(* IEC 61131-3 sources: rk/stdlib, 15 files *)

(* ---- Arrays.st ---- *)
/*
Array functions.

`LOWER_BOUND` and `UPPER_BOUND` read the bounds of an array. They take an
array of any type and any number of dimensions, so a FUNCTION with an
`ARRAY[*]` parameter can walk whatever array its caller passed.

`GET_DWORD_BE` and its siblings read a WORD, a DWORD, an LWORD, a REAL or an
LREAL out of an array of bytes, at a subscript of that array, in big-endian
(`_BE`) or little-endian (`_LE`) order. `PUT_DWORD_BE` and its siblings
write one. A position whose bytes are not all in the array faults, as any
subscript past its bounds does.
*/
NAMESPACE Std.Arrays

	/* Returns the lower bound of dimension `DIM` of `ARR`.

	   Dimensions are numbered from 1. A `DIM` outside them raises.

	   # Examples

	   ```iecst
	   FOR i := LOWER_BOUND(values, 1) TO UPPER_BOUND(values, 1) DO
	       total := total + values[i];
	   END_FOR;
	   ```
	*/
	FUNCTION LOWER_BOUND: DINT
		VAR_INPUT
			ARR: ARRAY[*];
			DIM: DINT;
		END_VAR
		VAR
			dimensions: DINT;
		END_VAR

		{wasm 'array.dimensions' (params ARR) (result dimensions)}
		IF DIM < 1 OR DIM > dimensions THEN
			__RAISE('array dimension out of range');
		END_IF
		{wasm 'array.lower_bound' (params ARR DIM) (result LOWER_BOUND)}
	END_FUNCTION

	/* Returns the upper bound of dimension `DIM` of `ARR`.

	   Dimensions are numbered from 1. A `DIM` outside them raises.

	   # Examples

	   ```iecst
	   // m : ARRAY[1..3, 0..9] OF REAL
	   rows := UPPER_BOUND(m, 1) - LOWER_BOUND(m, 1) + 1;     // 3
	   columns := UPPER_BOUND(m, 2) - LOWER_BOUND(m, 2) + 1;  // 10
	   ```
	*/
	FUNCTION UPPER_BOUND: DINT
		VAR_INPUT
			ARR: ARRAY[*];
			DIM: DINT;
		END_VAR
		VAR
			dimensions: DINT;
		END_VAR

		{wasm 'array.dimensions' (params ARR) (result dimensions)}
		IF DIM < 1 OR DIM > dimensions THEN
			__RAISE('array dimension out of range');
		END_IF
		{wasm 'array.upper_bound' (params ARR DIM) (result UPPER_BOUND)}
	END_FUNCTION

	/* Returns the value whose bytes are in `buf` from `pos` on, in big-endian
	   order: the most significant at `pos`.

	   # Examples

	   ```iecst
	   // frame holds 16#12, 16#34, 16#56, 16#78 from its subscript 0 on
	   d := GET_DWORD_BE(frame, 0);  // DWORD#16#12345678
	   w := GET_WORD_BE(frame, 2);   // WORD#16#5678
	   ```
	*/
	FUNCTION GET_WORD_BE: WORD
		VAR_IN_OUT
			buf: ARRAY[*] OF BYTE;
		END_VAR
		VAR_INPUT
			pos: DINT;
		END_VAR
		GET_WORD_BE.%B1 := buf[pos];
		GET_WORD_BE.%B0 := buf[pos + 1];
	END_FUNCTION

	FUNCTION GET_DWORD_BE: DWORD
		VAR_IN_OUT
			buf: ARRAY[*] OF BYTE;
		END_VAR
		VAR_INPUT
			pos: DINT;
		END_VAR
		GET_DWORD_BE.%B3 := buf[pos];
		GET_DWORD_BE.%B2 := buf[pos + 1];
		GET_DWORD_BE.%B1 := buf[pos + 2];
		GET_DWORD_BE.%B0 := buf[pos + 3];
	END_FUNCTION

	FUNCTION GET_LWORD_BE: LWORD
		VAR_IN_OUT
			buf: ARRAY[*] OF BYTE;
		END_VAR
		VAR_INPUT
			pos: DINT;
		END_VAR
		GET_LWORD_BE.%B7 := buf[pos];
		GET_LWORD_BE.%B6 := buf[pos + 1];
		GET_LWORD_BE.%B5 := buf[pos + 2];
		GET_LWORD_BE.%B4 := buf[pos + 3];
		GET_LWORD_BE.%B3 := buf[pos + 4];
		GET_LWORD_BE.%B2 := buf[pos + 5];
		GET_LWORD_BE.%B1 := buf[pos + 6];
		GET_LWORD_BE.%B0 := buf[pos + 7];
	END_FUNCTION

	FUNCTION GET_REAL_BE: REAL
		VAR_IN_OUT
			buf: ARRAY[*] OF BYTE;
		END_VAR
		VAR_INPUT
			pos: DINT;
		END_VAR
		VAR
			v: DWORD;
		END_VAR
		v := GET_DWORD_BE(buf, pos);
		{wasm 'f32.reinterpret_i32' (params v) (result GET_REAL_BE)}
	END_FUNCTION

	FUNCTION GET_LREAL_BE: LREAL
		VAR_IN_OUT
			buf: ARRAY[*] OF BYTE;
		END_VAR
		VAR_INPUT
			pos: DINT;
		END_VAR
		VAR
			v: LWORD;
		END_VAR
		v := GET_LWORD_BE(buf, pos);
		{wasm 'f64.reinterpret_i64' (params v) (result GET_LREAL_BE)}
	END_FUNCTION

	/* Returns the value whose bytes are in `buf` from `pos` on, in
	   little-endian order: the least significant at `pos`.

	   # Examples

	   ```iecst
	   // frame holds 16#12, 16#34, 16#56, 16#78 from its subscript 0 on
	   d := GET_DWORD_LE(frame, 0);  // DWORD#16#78563412
	   ```
	*/
	FUNCTION GET_WORD_LE: WORD
		VAR_IN_OUT
			buf: ARRAY[*] OF BYTE;
		END_VAR
		VAR_INPUT
			pos: DINT;
		END_VAR
		GET_WORD_LE.%B0 := buf[pos];
		GET_WORD_LE.%B1 := buf[pos + 1];
	END_FUNCTION

	FUNCTION GET_DWORD_LE: DWORD
		VAR_IN_OUT
			buf: ARRAY[*] OF BYTE;
		END_VAR
		VAR_INPUT
			pos: DINT;
		END_VAR
		GET_DWORD_LE.%B0 := buf[pos];
		GET_DWORD_LE.%B1 := buf[pos + 1];
		GET_DWORD_LE.%B2 := buf[pos + 2];
		GET_DWORD_LE.%B3 := buf[pos + 3];
	END_FUNCTION

	FUNCTION GET_LWORD_LE: LWORD
		VAR_IN_OUT
			buf: ARRAY[*] OF BYTE;
		END_VAR
		VAR_INPUT
			pos: DINT;
		END_VAR
		GET_LWORD_LE.%B0 := buf[pos];
		GET_LWORD_LE.%B1 := buf[pos + 1];
		GET_LWORD_LE.%B2 := buf[pos + 2];
		GET_LWORD_LE.%B3 := buf[pos + 3];
		GET_LWORD_LE.%B4 := buf[pos + 4];
		GET_LWORD_LE.%B5 := buf[pos + 5];
		GET_LWORD_LE.%B6 := buf[pos + 6];
		GET_LWORD_LE.%B7 := buf[pos + 7];
	END_FUNCTION

	FUNCTION GET_REAL_LE: REAL
		VAR_IN_OUT
			buf: ARRAY[*] OF BYTE;
		END_VAR
		VAR_INPUT
			pos: DINT;
		END_VAR
		VAR
			v: DWORD;
		END_VAR
		v := GET_DWORD_LE(buf, pos);
		{wasm 'f32.reinterpret_i32' (params v) (result GET_REAL_LE)}
	END_FUNCTION

	FUNCTION GET_LREAL_LE: LREAL
		VAR_IN_OUT
			buf: ARRAY[*] OF BYTE;
		END_VAR
		VAR_INPUT
			pos: DINT;
		END_VAR
		VAR
			v: LWORD;
		END_VAR
		v := GET_LWORD_LE(buf, pos);
		{wasm 'f64.reinterpret_i64' (params v) (result GET_LREAL_LE)}
	END_FUNCTION

	/* Writes the bytes of `value` into `buf` from `pos` on, in big-endian
	   order: the most significant at `pos`.

	   # Examples

	   ```iecst
	   PUT_DWORD_BE(frame, 0, DWORD#16#12345678);  // 16#12, 16#34, 16#56, 16#78
	   PUT_REAL_BE(frame, 4, REAL#1.0);            // 16#3F, 16#80, 16#00, 16#00
	   ```
	*/
	FUNCTION PUT_WORD_BE
		VAR_IN_OUT
			buf: ARRAY[*] OF BYTE;
		END_VAR
		VAR_INPUT
			pos: DINT;
			value: WORD;
		END_VAR
		buf[pos] := value.%B1;
		buf[pos + 1] := value.%B0;
	END_FUNCTION

	FUNCTION PUT_DWORD_BE
		VAR_IN_OUT
			buf: ARRAY[*] OF BYTE;
		END_VAR
		VAR_INPUT
			pos: DINT;
			value: DWORD;
		END_VAR
		buf[pos] := value.%B3;
		buf[pos + 1] := value.%B2;
		buf[pos + 2] := value.%B1;
		buf[pos + 3] := value.%B0;
	END_FUNCTION

	FUNCTION PUT_LWORD_BE
		VAR_IN_OUT
			buf: ARRAY[*] OF BYTE;
		END_VAR
		VAR_INPUT
			pos: DINT;
			value: LWORD;
		END_VAR
		buf[pos] := value.%B7;
		buf[pos + 1] := value.%B6;
		buf[pos + 2] := value.%B5;
		buf[pos + 3] := value.%B4;
		buf[pos + 4] := value.%B3;
		buf[pos + 5] := value.%B2;
		buf[pos + 6] := value.%B1;
		buf[pos + 7] := value.%B0;
	END_FUNCTION

	FUNCTION PUT_REAL_BE
		VAR_IN_OUT
			buf: ARRAY[*] OF BYTE;
		END_VAR
		VAR_INPUT
			pos: DINT;
			value: REAL;
		END_VAR
		VAR
			v: DWORD;
		END_VAR
		{wasm 'i32.reinterpret_f32' (params value) (result v)}
		PUT_DWORD_BE(buf, pos, v);
	END_FUNCTION

	FUNCTION PUT_LREAL_BE
		VAR_IN_OUT
			buf: ARRAY[*] OF BYTE;
		END_VAR
		VAR_INPUT
			pos: DINT;
			value: LREAL;
		END_VAR
		VAR
			v: LWORD;
		END_VAR
		{wasm 'i64.reinterpret_f64' (params value) (result v)}
		PUT_LWORD_BE(buf, pos, v);
	END_FUNCTION

	/* Writes the bytes of `value` into `buf` from `pos` on, in little-endian
	   order: the least significant at `pos`.

	   # Examples

	   ```iecst
	   PUT_DWORD_LE(frame, 0, DWORD#16#12345678);  // 16#78, 16#56, 16#34, 16#12
	   ```
	*/
	FUNCTION PUT_WORD_LE
		VAR_IN_OUT
			buf: ARRAY[*] OF BYTE;
		END_VAR
		VAR_INPUT
			pos: DINT;
			value: WORD;
		END_VAR
		buf[pos] := value.%B0;
		buf[pos + 1] := value.%B1;
	END_FUNCTION

	FUNCTION PUT_DWORD_LE
		VAR_IN_OUT
			buf: ARRAY[*] OF BYTE;
		END_VAR
		VAR_INPUT
			pos: DINT;
			value: DWORD;
		END_VAR
		buf[pos] := value.%B0;
		buf[pos + 1] := value.%B1;
		buf[pos + 2] := value.%B2;
		buf[pos + 3] := value.%B3;
	END_FUNCTION

	FUNCTION PUT_LWORD_LE
		VAR_IN_OUT
			buf: ARRAY[*] OF BYTE;
		END_VAR
		VAR_INPUT
			pos: DINT;
			value: LWORD;
		END_VAR
		buf[pos] := value.%B0;
		buf[pos + 1] := value.%B1;
		buf[pos + 2] := value.%B2;
		buf[pos + 3] := value.%B3;
		buf[pos + 4] := value.%B4;
		buf[pos + 5] := value.%B5;
		buf[pos + 6] := value.%B6;
		buf[pos + 7] := value.%B7;
	END_FUNCTION

	FUNCTION PUT_REAL_LE
		VAR_IN_OUT
			buf: ARRAY[*] OF BYTE;
		END_VAR
		VAR_INPUT
			pos: DINT;
			value: REAL;
		END_VAR
		VAR
			v: DWORD;
		END_VAR
		{wasm 'i32.reinterpret_f32' (params value) (result v)}
		PUT_DWORD_LE(buf, pos, v);
	END_FUNCTION

	FUNCTION PUT_LREAL_LE
		VAR_IN_OUT
			buf: ARRAY[*] OF BYTE;
		END_VAR
		VAR_INPUT
			pos: DINT;
			value: LREAL;
		END_VAR
		VAR
			v: LWORD;
		END_VAR
		{wasm 'i64.reinterpret_f64' (params value) (result v)}
		PUT_LWORD_LE(buf, pos, v);
	END_FUNCTION

	NAMESPACE Test
		USING Std.Unit

		{test}
		FUNCTION test_bounds_of_one_dimension
			VAR
				a: ARRAY[1..10] OF INT;
			END_VAR
			ASSERT(LOWER_BOUND(a, 1) = 1 AND UPPER_BOUND(a, 1) = 10);
		END_FUNCTION

		{test}
		FUNCTION test_bounds_of_each_dimension
			VAR
				a: ARRAY[1..20, -2..2] OF INT;
			END_VAR
			ASSERT(LOWER_BOUND(a, 1) = 1 AND UPPER_BOUND(a, 1) = 20);
			ASSERT(LOWER_BOUND(a, 2) = -2 AND UPPER_BOUND(a, 2) = 2);
		END_FUNCTION

		{test}
		FUNCTION test_bounds_by_name
			VAR
				a: ARRAY[5..7] OF STRING[4];
			END_VAR
			ASSERT(LOWER_BOUND(ARR := a, DIM := 1) = 5);
			ASSERT(UPPER_BOUND(DIM := 1, ARR := a) = 7);
		END_FUNCTION

		FUNCTION Sum: DINT
			VAR_IN_OUT
				values: ARRAY[*] OF INT;
			END_VAR
			VAR
				i: DINT;
			END_VAR
			FOR i := LOWER_BOUND(values, 1) TO UPPER_BOUND(values, 1) DO
				Sum := Sum + values[i];
			END_FOR
		END_FUNCTION

		{test}
		FUNCTION test_bounds_of_an_array_any_call_binds
			VAR
				a: ARRAY[1..20, -2..2] OF INT := [20(5(1))];
				b: ARRAY[0..2] OF INT := [1, 2, 3];
			END_VAR
			ASSERT(Sum(a[2]) = 5, 'a row of a');
			ASSERT(Sum(b) = 6, 'b');
		END_FUNCTION

		{test}
		FUNCTION test_get_word_be
			VAR b : ARRAY[0..1] OF BYTE := [16#12, 16#34]; END_VAR
			ASSERT_EQ(GET_WORD_BE(b, 0), WORD#16#1234);
		END_FUNCTION

		{test}
		FUNCTION test_get_word_le
			VAR b : ARRAY[0..1] OF BYTE := [16#12, 16#34]; END_VAR
			ASSERT_EQ(GET_WORD_LE(b, 0), WORD#16#3412);
		END_FUNCTION

		{test}
		FUNCTION test_get_dword_at_a_subscript
			VAR b : ARRAY[1..6] OF BYTE := [16#FF, 16#12, 16#34, 16#56, 16#78, 16#FF]; END_VAR
			ASSERT_EQ(GET_DWORD_BE(b, 2), DWORD#16#12345678);
		END_FUNCTION

		{test}
		FUNCTION test_put_dword_be
			VAR b : ARRAY[0..3] OF BYTE; END_VAR
			PUT_DWORD_BE(b, 0, DWORD#16#12345678);
			ASSERT_EQ(b[0], BYTE#16#12);
			ASSERT_EQ(b[3], BYTE#16#78);
		END_FUNCTION

		{test}
		FUNCTION test_put_dword_le
			VAR b : ARRAY[0..3] OF BYTE; END_VAR
			PUT_DWORD_LE(b, 0, DWORD#16#12345678);
			ASSERT_EQ(b[0], BYTE#16#78);
			ASSERT_EQ(b[3], BYTE#16#12);
		END_FUNCTION

		{test}
		FUNCTION test_lword_round_trip
			VAR b : ARRAY[0..9] OF BYTE; END_VAR
			PUT_LWORD_BE(b, 1, LWORD#16#0102030405060708);
			ASSERT_EQ(b[1], BYTE#16#01);
			ASSERT_EQ(b[8], BYTE#16#08);
			ASSERT_EQ(GET_LWORD_BE(b, 1), LWORD#16#0102030405060708);
			ASSERT_EQ(GET_LWORD_LE(b, 1), LWORD#16#0807060504030201);
		END_FUNCTION

		{test}
		FUNCTION test_put_real_be
			VAR b : ARRAY[0..3] OF BYTE; END_VAR
			PUT_REAL_BE(b, 0, REAL#1.0);
			ASSERT_EQ(b[0], BYTE#16#3F);
			ASSERT_EQ(b[1], BYTE#16#80);
			ASSERT_EQ(GET_REAL_BE(b, 0), REAL#1.0);
		END_FUNCTION

		{test}
		FUNCTION test_real_le_round_trip
			VAR b : ARRAY[0..3] OF BYTE; END_VAR
			PUT_REAL_LE(b, 0, REAL#-2.5);
			ASSERT_EQ(b[3], BYTE#16#C0);
			ASSERT_EQ(GET_REAL_LE(b, 0), REAL#-2.5);
		END_FUNCTION

		{test}
		FUNCTION test_put_lreal_be
			VAR b : ARRAY[0..7] OF BYTE; END_VAR
			PUT_LREAL_BE(b, 0, LREAL#1.5);
			ASSERT_EQ(b[0], BYTE#16#3F);
			ASSERT_EQ(b[1], BYTE#16#F8);
			ASSERT_EQ(GET_LREAL_BE(b, 0), LREAL#1.5);
		END_FUNCTION

		{test}
		FUNCTION test_lreal_le_round_trip
			VAR b : ARRAY[0..7] OF BYTE; END_VAR
			PUT_LREAL_LE(b, 0, LREAL#1.5);
			ASSERT_EQ(b[7], BYTE#16#3F);
			ASSERT_EQ(GET_LREAL_LE(b, 0), LREAL#1.5);
		END_FUNCTION
	END_NAMESPACE

END_NAMESPACE

(* ---- Bits.st ---- *)
/*
Bit shift and rotate functions.

Each takes a `BYTE`, `WORD`, `DWORD` or `LWORD` and a count `N`, and returns
the type it was given. The width is that of the type: a `BYTE` is shifted
and rotated within its 8 bits.
*/
NAMESPACE Std.Bits

	/* Returns `IN` shifted left by `N` bits, filling with zeros.

	   Bits shifted past the top of the type are lost. An `N` of the type's width
	   or more gives 0.

	   # Examples

	   ```iecst
	   b := SHL(BYTE#16#0F, 4);    // BYTE#16#F0
	   b := SHL(BYTE#16#FF, 4);    // BYTE#16#F0
	   w := SHL(WORD#16#0001, 8);  // WORD#16#0100
	   b := SHL(BYTE#16#01, 8);    // BYTE#16#00
	   ```
	*/
	FUNCTION SHL: BYTE
		VAR_INPUT
			IN: BYTE;
			N: INT;
		END_VAR
		{wasm IN 'shl' (params IN N) (result SHL)}
	END_FUNCTION

	FUNCTION SHL: WORD
		VAR_INPUT
			IN: WORD;
			N: INT;
		END_VAR
		{wasm IN 'shl' (params IN N) (result SHL)}
	END_FUNCTION

	FUNCTION SHL: DWORD
		VAR_INPUT
			IN: DWORD;
			N: INT;
		END_VAR
		{wasm IN 'shl' (params IN N) (result SHL)}
	END_FUNCTION

	FUNCTION SHL: LWORD
		VAR_INPUT
			IN: LWORD;
			N: INT;
		END_VAR
		{wasm IN 'shl' (params IN N) (result SHL)}
	END_FUNCTION

	/* Returns `IN` shifted right by `N` bits, filling with zeros.

	   An `N` of the type's width or more gives 0.

	   # Examples

	   ```iecst
	   b := SHR(BYTE#16#F0, 4);         // BYTE#16#0F
	   d := SHR(DWORD#16#80000000, 31);  // DWORD#1
	   ```
	*/
	FUNCTION SHR: BYTE
		VAR_INPUT
			IN: BYTE;
			N: INT;
		END_VAR
		{wasm IN 'shr_u' (params IN N) (result SHR)}
	END_FUNCTION

	FUNCTION SHR: WORD
		VAR_INPUT
			IN: WORD;
			N: INT;
		END_VAR
		{wasm IN 'shr_u' (params IN N) (result SHR)}
	END_FUNCTION

	FUNCTION SHR: DWORD
		VAR_INPUT
			IN: DWORD;
			N: INT;
		END_VAR
		{wasm IN 'shr_u' (params IN N) (result SHR)}
	END_FUNCTION

	FUNCTION SHR: LWORD
		VAR_INPUT
			IN: LWORD;
			N: INT;
		END_VAR
		{wasm IN 'shr_u' (params IN N) (result SHR)}
	END_FUNCTION

	/* Returns `IN` rotated left by `N` bits.

	   Bits that leave at the top come back at the bottom. `N` wraps at the type's
	   width, so rotating a `BYTE` by 8 returns it unchanged.

	   # Examples

	   ```iecst
	   b := ROL(BYTE#16#81, 1);  // BYTE#16#03
	   b := ROL(BYTE#16#81, 8);  // BYTE#16#81
	   ```
	*/
	FUNCTION ROL: BYTE
		VAR_INPUT
			IN: BYTE;
			N: INT;
		END_VAR
		{wasm IN 'rotl' (params IN N) (result ROL)}
	END_FUNCTION

	FUNCTION ROL: WORD
		VAR_INPUT
			IN: WORD;
			N: INT;
		END_VAR
		{wasm IN 'rotl' (params IN N) (result ROL)}
	END_FUNCTION

	FUNCTION ROL: DWORD
		VAR_INPUT
			IN: DWORD;
			N: INT;
		END_VAR
		{wasm IN 'rotl' (params IN N) (result ROL)}
	END_FUNCTION

	FUNCTION ROL: LWORD
		VAR_INPUT
			IN: LWORD;
			N: INT;
		END_VAR
		{wasm IN 'rotl' (params IN N) (result ROL)}
	END_FUNCTION

	/* Returns `IN` rotated right by `N` bits.

	   Bits that leave at the bottom come back at the top. `N` wraps at the type's
	   width.

	   # Examples

	   ```iecst
	   b := ROR(BYTE#16#01, 1);  // BYTE#16#80
	   w := ROR(WORD#16#0001, 1);  // WORD#16#8000
	   ```
	*/
	FUNCTION ROR: BYTE
		VAR_INPUT
			IN: BYTE;
			N: INT;
		END_VAR
		{wasm IN 'rotr' (params IN N) (result ROR)}
	END_FUNCTION

	FUNCTION ROR: WORD
		VAR_INPUT
			IN: WORD;
			N: INT;
		END_VAR
		{wasm IN 'rotr' (params IN N) (result ROR)}
	END_FUNCTION

	FUNCTION ROR: DWORD
		VAR_INPUT
			IN: DWORD;
			N: INT;
		END_VAR
		{wasm IN 'rotr' (params IN N) (result ROR)}
	END_FUNCTION

	FUNCTION ROR: LWORD
		VAR_INPUT
			IN: LWORD;
			N: INT;
		END_VAR
		{wasm IN 'rotr' (params IN N) (result ROR)}
	END_FUNCTION

	NAMESPACE Test
		USING Std.Unit

		{test}
		FUNCTION test_shl_byte ASSERT_EQ(SHL(BYTE#16#0F, 4), BYTE#16#F0);
		END_FUNCTION

		{test}
		FUNCTION test_shr_byte ASSERT_EQ(SHR(BYTE#16#F0, 4), BYTE#16#0F);
		END_FUNCTION

		{test}
		FUNCTION test_shl_word ASSERT_EQ(SHL(WORD#16#0001, 8), WORD#16#0100);
		END_FUNCTION

		{test}
		FUNCTION test_shr_word ASSERT_EQ(SHR(WORD#16#0100, 8), WORD#16#0001);
		END_FUNCTION

		{test}
		FUNCTION test_rol_dword ASSERT_EQ(ROL(DWORD#1, 4), DWORD#16);
		END_FUNCTION

		{test}
		FUNCTION test_ror_dword ASSERT_EQ(ROR(DWORD#16, 4), DWORD#1);
		END_FUNCTION

		// --- edge cases ---

		// Shift/rotate by 0 is the identity, independent of storage width.
		{test}
		FUNCTION test_shl_by_zero ASSERT_EQ(SHL(BYTE#16#0F, 0), BYTE#16#0F);
		END_FUNCTION

		{test}
		FUNCTION test_shr_by_zero ASSERT_EQ(SHR(WORD#16#00F0, 0), WORD#16#00F0);
		END_FUNCTION

		{test}
		FUNCTION test_rol_by_zero ASSERT_EQ(ROL(DWORD#16#12345678, 0), DWORD#16#12345678);
		END_FUNCTION

		{test}
		FUNCTION test_ror_by_zero ASSERT_EQ(ROR(DWORD#16#12345678, 0), DWORD#16#12345678);
		END_FUNCTION

		// DWORD is i32-backed, so rotate wraps correctly at 32 bits:
		// the top bit rotated left re-enters at bit 0.
		{test}
		FUNCTION test_rol_dword_wraps_msb ASSERT_EQ(ROL(DWORD#16#80000000, 1), DWORD#1);
		END_FUNCTION

		{test}
		FUNCTION test_ror_dword_wraps_lsb ASSERT_EQ(ROR(DWORD#1, 1), DWORD#16#80000000);
		END_FUNCTION

		// Logical shift right fills with zeros (no sign extension) on a bit type.
		{test}
		FUNCTION test_shr_dword_top_bit ASSERT_EQ(SHR(DWORD#16#80000000, 31), DWORD#1);
		END_FUNCTION

		// --- sub-width masking: shifted-out bits must not leak past the type width ---

		{test}
		FUNCTION test_shl_byte_masks_leak
			ASSERT_EQ(SHL(BYTE#16#FF, 4), BYTE#16#F0, 'SHL BYTE must mask bits above bit 7');
		END_FUNCTION

		{test}
		FUNCTION test_shl_word_masks_leak
			ASSERT_EQ(SHL(WORD#16#FFFF, 8), WORD#16#FF00, 'SHL WORD must mask bits above bit 15');
		END_FUNCTION

		{test}
		FUNCTION test_shl_byte_by_type_width
			ASSERT_EQ(SHL(BYTE#16#01, 8), BYTE#16#00, 'shift by the full type width empties the value');
		END_FUNCTION

		// --- shift count >= width yields 0 (wasm masks the count mod the lane
		// width, so a raw lowering would return the input unchanged) ---

		{test}
		FUNCTION test_shl_dword_by_32
			ASSERT_EQ(SHL(DWORD#1, 32), DWORD#0, 'SHL DWORD by 32 is 0, not a wasm count-mask no-op');
		END_FUNCTION

		{test}
		FUNCTION test_shr_dword_by_32
			ASSERT_EQ(SHR(DWORD#16#80000000, 32), DWORD#0, 'SHR DWORD by 32 is 0');
		END_FUNCTION

		{test}
		FUNCTION test_shr_word_by_32
			ASSERT_EQ(SHR(WORD#16#0001, 32), WORD#0, 'SHR WORD by 32 hits the wasm lane mask');
		END_FUNCTION

		// --- sub-width rotates wrap at the type MSB/LSB, not bit 31 ---

		{test}
		FUNCTION test_rol_byte_wraps_msb
			// The doc example: the wrapped bit re-enters at bit 0, not bit 8.
			ASSERT_EQ(ROL(BYTE#16#81, 1), BYTE#16#03, 'ROL BYTE MSB wraps to bit 0');
		END_FUNCTION

		{test}
		FUNCTION test_ror_byte_wraps_lsb
			ASSERT_EQ(ROR(BYTE#16#01, 1), BYTE#16#80, 'ROR BYTE LSB wraps to bit 7, not bit 31');
		END_FUNCTION

		{test}
		FUNCTION test_rol_word_wraps_msb
			ASSERT_EQ(ROL(WORD#16#8001, 1), WORD#16#0003, 'ROL WORD bit 15 wraps to bit 0');
		END_FUNCTION

		{test}
		FUNCTION test_ror_word_wraps_lsb
			ASSERT_EQ(ROR(WORD#16#0001, 1), WORD#16#8000, 'ROR WORD LSB wraps to bit 15');
		END_FUNCTION

		// Rotate counts are mod the type width.
		{test}
		FUNCTION test_rol_byte_count_mod_width
			ASSERT_EQ(ROL(BYTE#16#81, 0), BYTE#16#81, 'ROL by 0 is identity');
			ASSERT_EQ(ROL(BYTE#16#81, 8), BYTE#16#81, 'ROL by the type width is identity');
			ASSERT_EQ(ROL(BYTE#16#81, 9), BYTE#16#03, 'ROL by 9 = ROL by 1 (mod 8)');
		END_FUNCTION

		// --- LWORD (i64 lane): value, count extension, and 64-bit wraps ---

		{test}
		FUNCTION test_shl_lword_crosses_32
			ASSERT_EQ(SHL(LWORD#1, 32), LWORD#16#0000_0001_0000_0000, 'SHL LWORD must cross the 32-bit line');
		END_FUNCTION

		{test}
		FUNCTION test_shl_lword_by_64
			ASSERT_EQ(SHL(LWORD#1, 64), LWORD#0, 'SHL LWORD by 64 is 0');
		END_FUNCTION

		{test}
		FUNCTION test_shr_lword_top_bit
			ASSERT_EQ(SHR(LWORD#16#8000_0000_0000_0000, 63), LWORD#1, 'logical shift on the i64 lane');
		END_FUNCTION

		{test}
		FUNCTION test_rol_lword_wraps_msb
			ASSERT_EQ(ROL(LWORD#16#8000_0000_0000_0000, 1), LWORD#1, '64-bit MSB wraps to bit 0');
		END_FUNCTION

		{test}
		FUNCTION test_ror_lword_wraps_lsb
			ASSERT_EQ(ROR(LWORD#1, 1), LWORD#16#8000_0000_0000_0000, '64-bit LSB wraps to bit 63');
		END_FUNCTION

		{test}
		FUNCTION test_shr_byte_after_shl_roundtrip
			// SHR on a sub-width type relies on the masked-value invariant.
			ASSERT_EQ(SHR(SHL(BYTE#16#FF, 4), 4), BYTE#16#0F, 'SHL then SHR keeps only surviving bits');
		END_FUNCTION
	END_NAMESPACE
END_NAMESPACE

(* ---- Bytes.st ---- *)
/*
Byte order and BCD.

rk keeps every value in little-endian order, the order of WebAssembly: its
least significant byte at the lowest address. TO_BIG_ENDIAN and
FROM_BIG_ENDIAN reverse the bytes of a value, and TO_LITTLE_ENDIAN and
FROM_LITTLE_ENDIAN return it as it is.

Each takes an integer, a bit string, a REAL, an LREAL, a TIME or an LTIME,
and returns the type it was given. A value of one byte has no order, and is
returned as it is.

BCD stores a number one decimal digit in each 4 bits: WORD#16#0369 is 369.
Its conversions go between a bit string and the unsigned integer of the same
width, from BYTE and USINT to LWORD and ULINT.
*/
NAMESPACE Std.Bytes

	/* Returns `IN` with its bytes in big-endian order, the most significant
	   first: the order a peer reading big-endian data expects.

	   # Examples

	   ```iecst
	   w := TO_BIG_ENDIAN(WORD#16#1234);       // WORD#16#3412
	   d := TO_BIG_ENDIAN(DWORD#16#12345678);  // DWORD#16#78563412
	   b := TO_BIG_ENDIAN(BYTE#16#AB);         // BYTE#16#AB
	   ```
	*/
	FUNCTION TO_BIG_ENDIAN: BYTE
		VAR_INPUT
			IN: BYTE;
		END_VAR
		TO_BIG_ENDIAN := IN;
	END_FUNCTION

	FUNCTION TO_BIG_ENDIAN: SINT
		VAR_INPUT
			IN: SINT;
		END_VAR
		TO_BIG_ENDIAN := IN;
	END_FUNCTION

	FUNCTION TO_BIG_ENDIAN: USINT
		VAR_INPUT
			IN: USINT;
		END_VAR
		TO_BIG_ENDIAN := IN;
	END_FUNCTION

	FUNCTION TO_BIG_ENDIAN: WORD
		VAR_INPUT
			IN: WORD;
		END_VAR
		{wasm IN 'bswap' (params IN) (result TO_BIG_ENDIAN)}
	END_FUNCTION

	FUNCTION TO_BIG_ENDIAN: INT
		VAR_INPUT
			IN: INT;
		END_VAR
		VAR
			swapped: WORD;
		END_VAR
		{wasm IN 'bswap' (params IN) (result swapped)}
		{wasm 'nop' (params swapped) (result TO_BIG_ENDIAN)}
	END_FUNCTION

	FUNCTION TO_BIG_ENDIAN: UINT
		VAR_INPUT
			IN: UINT;
		END_VAR
		{wasm IN 'bswap' (params IN) (result TO_BIG_ENDIAN)}
	END_FUNCTION

	FUNCTION TO_BIG_ENDIAN: DWORD
		VAR_INPUT
			IN: DWORD;
		END_VAR
		{wasm IN 'bswap' (params IN) (result TO_BIG_ENDIAN)}
	END_FUNCTION

	FUNCTION TO_BIG_ENDIAN: DINT
		VAR_INPUT
			IN: DINT;
		END_VAR
		{wasm IN 'bswap' (params IN) (result TO_BIG_ENDIAN)}
	END_FUNCTION

	FUNCTION TO_BIG_ENDIAN: UDINT
		VAR_INPUT
			IN: UDINT;
		END_VAR
		{wasm IN 'bswap' (params IN) (result TO_BIG_ENDIAN)}
	END_FUNCTION

	FUNCTION TO_BIG_ENDIAN: REAL
		VAR_INPUT
			IN: REAL;
		END_VAR
		VAR
			bits: DWORD;
		END_VAR
		{wasm 'i32.reinterpret_f32' (params IN) (result bits)}
		{wasm bits 'bswap' (params bits) (result bits)}
		{wasm 'f32.reinterpret_i32' (params bits) (result TO_BIG_ENDIAN)}
	END_FUNCTION

	FUNCTION TO_BIG_ENDIAN: TIME
		VAR_INPUT
			IN: TIME;
		END_VAR
		{wasm IN 'bswap' (params IN) (result TO_BIG_ENDIAN)}
	END_FUNCTION

	FUNCTION TO_BIG_ENDIAN: LWORD
		VAR_INPUT
			IN: LWORD;
		END_VAR
		{wasm IN 'bswap' (params IN) (result TO_BIG_ENDIAN)}
	END_FUNCTION

	FUNCTION TO_BIG_ENDIAN: LINT
		VAR_INPUT
			IN: LINT;
		END_VAR
		{wasm IN 'bswap' (params IN) (result TO_BIG_ENDIAN)}
	END_FUNCTION

	FUNCTION TO_BIG_ENDIAN: ULINT
		VAR_INPUT
			IN: ULINT;
		END_VAR
		{wasm IN 'bswap' (params IN) (result TO_BIG_ENDIAN)}
	END_FUNCTION

	FUNCTION TO_BIG_ENDIAN: LREAL
		VAR_INPUT
			IN: LREAL;
		END_VAR
		VAR
			bits: LWORD;
		END_VAR
		{wasm 'i64.reinterpret_f64' (params IN) (result bits)}
		{wasm bits 'bswap' (params bits) (result bits)}
		{wasm 'f64.reinterpret_i64' (params bits) (result TO_BIG_ENDIAN)}
	END_FUNCTION

	FUNCTION TO_BIG_ENDIAN: LTIME
		VAR_INPUT
			IN: LTIME;
		END_VAR
		{wasm IN 'bswap' (params IN) (result TO_BIG_ENDIAN)}
	END_FUNCTION

	/* Returns `IN`, whose bytes are in big-endian order, in the order rk
	   computes with.

	   # Examples

	   ```iecst
	   w := FROM_BIG_ENDIAN(WORD#16#3412);     // WORD#16#1234
	   ```
	*/
	FUNCTION FROM_BIG_ENDIAN: BYTE
		VAR_INPUT
			IN: BYTE;
		END_VAR
		FROM_BIG_ENDIAN := IN;
	END_FUNCTION

	FUNCTION FROM_BIG_ENDIAN: SINT
		VAR_INPUT
			IN: SINT;
		END_VAR
		FROM_BIG_ENDIAN := IN;
	END_FUNCTION

	FUNCTION FROM_BIG_ENDIAN: USINT
		VAR_INPUT
			IN: USINT;
		END_VAR
		FROM_BIG_ENDIAN := IN;
	END_FUNCTION

	FUNCTION FROM_BIG_ENDIAN: WORD
		VAR_INPUT
			IN: WORD;
		END_VAR
		{wasm IN 'bswap' (params IN) (result FROM_BIG_ENDIAN)}
	END_FUNCTION

	FUNCTION FROM_BIG_ENDIAN: INT
		VAR_INPUT
			IN: INT;
		END_VAR
		VAR
			swapped: WORD;
		END_VAR
		{wasm IN 'bswap' (params IN) (result swapped)}
		{wasm 'nop' (params swapped) (result FROM_BIG_ENDIAN)}
	END_FUNCTION

	FUNCTION FROM_BIG_ENDIAN: UINT
		VAR_INPUT
			IN: UINT;
		END_VAR
		{wasm IN 'bswap' (params IN) (result FROM_BIG_ENDIAN)}
	END_FUNCTION

	FUNCTION FROM_BIG_ENDIAN: DWORD
		VAR_INPUT
			IN: DWORD;
		END_VAR
		{wasm IN 'bswap' (params IN) (result FROM_BIG_ENDIAN)}
	END_FUNCTION

	FUNCTION FROM_BIG_ENDIAN: DINT
		VAR_INPUT
			IN: DINT;
		END_VAR
		{wasm IN 'bswap' (params IN) (result FROM_BIG_ENDIAN)}
	END_FUNCTION

	FUNCTION FROM_BIG_ENDIAN: UDINT
		VAR_INPUT
			IN: UDINT;
		END_VAR
		{wasm IN 'bswap' (params IN) (result FROM_BIG_ENDIAN)}
	END_FUNCTION

	FUNCTION FROM_BIG_ENDIAN: REAL
		VAR_INPUT
			IN: REAL;
		END_VAR
		VAR
			bits: DWORD;
		END_VAR
		{wasm 'i32.reinterpret_f32' (params IN) (result bits)}
		{wasm bits 'bswap' (params bits) (result bits)}
		{wasm 'f32.reinterpret_i32' (params bits) (result FROM_BIG_ENDIAN)}
	END_FUNCTION

	FUNCTION FROM_BIG_ENDIAN: TIME
		VAR_INPUT
			IN: TIME;
		END_VAR
		{wasm IN 'bswap' (params IN) (result FROM_BIG_ENDIAN)}
	END_FUNCTION

	FUNCTION FROM_BIG_ENDIAN: LWORD
		VAR_INPUT
			IN: LWORD;
		END_VAR
		{wasm IN 'bswap' (params IN) (result FROM_BIG_ENDIAN)}
	END_FUNCTION

	FUNCTION FROM_BIG_ENDIAN: LINT
		VAR_INPUT
			IN: LINT;
		END_VAR
		{wasm IN 'bswap' (params IN) (result FROM_BIG_ENDIAN)}
	END_FUNCTION

	FUNCTION FROM_BIG_ENDIAN: ULINT
		VAR_INPUT
			IN: ULINT;
		END_VAR
		{wasm IN 'bswap' (params IN) (result FROM_BIG_ENDIAN)}
	END_FUNCTION

	FUNCTION FROM_BIG_ENDIAN: LREAL
		VAR_INPUT
			IN: LREAL;
		END_VAR
		VAR
			bits: LWORD;
		END_VAR
		{wasm 'i64.reinterpret_f64' (params IN) (result bits)}
		{wasm bits 'bswap' (params bits) (result bits)}
		{wasm 'f64.reinterpret_i64' (params bits) (result FROM_BIG_ENDIAN)}
	END_FUNCTION

	FUNCTION FROM_BIG_ENDIAN: LTIME
		VAR_INPUT
			IN: LTIME;
		END_VAR
		{wasm IN 'bswap' (params IN) (result FROM_BIG_ENDIAN)}
	END_FUNCTION

	/* Returns `IN` with its bytes in little-endian order, the least
	   significant first. rk keeps every value in that order, so `IN` is
	   returned as it is.
	*/
	FUNCTION TO_LITTLE_ENDIAN: BYTE
		VAR_INPUT
			IN: BYTE;
		END_VAR
		TO_LITTLE_ENDIAN := IN;
	END_FUNCTION

	FUNCTION TO_LITTLE_ENDIAN: SINT
		VAR_INPUT
			IN: SINT;
		END_VAR
		TO_LITTLE_ENDIAN := IN;
	END_FUNCTION

	FUNCTION TO_LITTLE_ENDIAN: USINT
		VAR_INPUT
			IN: USINT;
		END_VAR
		TO_LITTLE_ENDIAN := IN;
	END_FUNCTION

	FUNCTION TO_LITTLE_ENDIAN: WORD
		VAR_INPUT
			IN: WORD;
		END_VAR
		TO_LITTLE_ENDIAN := IN;
	END_FUNCTION

	FUNCTION TO_LITTLE_ENDIAN: INT
		VAR_INPUT
			IN: INT;
		END_VAR
		TO_LITTLE_ENDIAN := IN;
	END_FUNCTION

	FUNCTION TO_LITTLE_ENDIAN: UINT
		VAR_INPUT
			IN: UINT;
		END_VAR
		TO_LITTLE_ENDIAN := IN;
	END_FUNCTION

	FUNCTION TO_LITTLE_ENDIAN: DWORD
		VAR_INPUT
			IN: DWORD;
		END_VAR
		TO_LITTLE_ENDIAN := IN;
	END_FUNCTION

	FUNCTION TO_LITTLE_ENDIAN: DINT
		VAR_INPUT
			IN: DINT;
		END_VAR
		TO_LITTLE_ENDIAN := IN;
	END_FUNCTION

	FUNCTION TO_LITTLE_ENDIAN: UDINT
		VAR_INPUT
			IN: UDINT;
		END_VAR
		TO_LITTLE_ENDIAN := IN;
	END_FUNCTION

	FUNCTION TO_LITTLE_ENDIAN: REAL
		VAR_INPUT
			IN: REAL;
		END_VAR
		TO_LITTLE_ENDIAN := IN;
	END_FUNCTION

	FUNCTION TO_LITTLE_ENDIAN: TIME
		VAR_INPUT
			IN: TIME;
		END_VAR
		TO_LITTLE_ENDIAN := IN;
	END_FUNCTION

	FUNCTION TO_LITTLE_ENDIAN: LWORD
		VAR_INPUT
			IN: LWORD;
		END_VAR
		TO_LITTLE_ENDIAN := IN;
	END_FUNCTION

	FUNCTION TO_LITTLE_ENDIAN: LINT
		VAR_INPUT
			IN: LINT;
		END_VAR
		TO_LITTLE_ENDIAN := IN;
	END_FUNCTION

	FUNCTION TO_LITTLE_ENDIAN: ULINT
		VAR_INPUT
			IN: ULINT;
		END_VAR
		TO_LITTLE_ENDIAN := IN;
	END_FUNCTION

	FUNCTION TO_LITTLE_ENDIAN: LREAL
		VAR_INPUT
			IN: LREAL;
		END_VAR
		TO_LITTLE_ENDIAN := IN;
	END_FUNCTION

	FUNCTION TO_LITTLE_ENDIAN: LTIME
		VAR_INPUT
			IN: LTIME;
		END_VAR
		TO_LITTLE_ENDIAN := IN;
	END_FUNCTION

	/* Returns `IN`, whose bytes are in little-endian order, in the order rk
	   computes with. rk keeps every value in that order, so `IN` is
	   returned as it is.
	*/
	FUNCTION FROM_LITTLE_ENDIAN: BYTE
		VAR_INPUT
			IN: BYTE;
		END_VAR
		FROM_LITTLE_ENDIAN := IN;
	END_FUNCTION

	FUNCTION FROM_LITTLE_ENDIAN: SINT
		VAR_INPUT
			IN: SINT;
		END_VAR
		FROM_LITTLE_ENDIAN := IN;
	END_FUNCTION

	FUNCTION FROM_LITTLE_ENDIAN: USINT
		VAR_INPUT
			IN: USINT;
		END_VAR
		FROM_LITTLE_ENDIAN := IN;
	END_FUNCTION

	FUNCTION FROM_LITTLE_ENDIAN: WORD
		VAR_INPUT
			IN: WORD;
		END_VAR
		FROM_LITTLE_ENDIAN := IN;
	END_FUNCTION

	FUNCTION FROM_LITTLE_ENDIAN: INT
		VAR_INPUT
			IN: INT;
		END_VAR
		FROM_LITTLE_ENDIAN := IN;
	END_FUNCTION

	FUNCTION FROM_LITTLE_ENDIAN: UINT
		VAR_INPUT
			IN: UINT;
		END_VAR
		FROM_LITTLE_ENDIAN := IN;
	END_FUNCTION

	FUNCTION FROM_LITTLE_ENDIAN: DWORD
		VAR_INPUT
			IN: DWORD;
		END_VAR
		FROM_LITTLE_ENDIAN := IN;
	END_FUNCTION

	FUNCTION FROM_LITTLE_ENDIAN: DINT
		VAR_INPUT
			IN: DINT;
		END_VAR
		FROM_LITTLE_ENDIAN := IN;
	END_FUNCTION

	FUNCTION FROM_LITTLE_ENDIAN: UDINT
		VAR_INPUT
			IN: UDINT;
		END_VAR
		FROM_LITTLE_ENDIAN := IN;
	END_FUNCTION

	FUNCTION FROM_LITTLE_ENDIAN: REAL
		VAR_INPUT
			IN: REAL;
		END_VAR
		FROM_LITTLE_ENDIAN := IN;
	END_FUNCTION

	FUNCTION FROM_LITTLE_ENDIAN: TIME
		VAR_INPUT
			IN: TIME;
		END_VAR
		FROM_LITTLE_ENDIAN := IN;
	END_FUNCTION

	FUNCTION FROM_LITTLE_ENDIAN: LWORD
		VAR_INPUT
			IN: LWORD;
		END_VAR
		FROM_LITTLE_ENDIAN := IN;
	END_FUNCTION

	FUNCTION FROM_LITTLE_ENDIAN: LINT
		VAR_INPUT
			IN: LINT;
		END_VAR
		FROM_LITTLE_ENDIAN := IN;
	END_FUNCTION

	FUNCTION FROM_LITTLE_ENDIAN: ULINT
		VAR_INPUT
			IN: ULINT;
		END_VAR
		FROM_LITTLE_ENDIAN := IN;
	END_FUNCTION

	FUNCTION FROM_LITTLE_ENDIAN: LREAL
		VAR_INPUT
			IN: LREAL;
		END_VAR
		FROM_LITTLE_ENDIAN := IN;
	END_FUNCTION

	FUNCTION FROM_LITTLE_ENDIAN: LTIME
		VAR_INPUT
			IN: LTIME;
		END_VAR
		FROM_LITTLE_ENDIAN := IN;
	END_FUNCTION

	/* Returns the number `IN` holds in BCD, one decimal digit in each 4 bits,
	   the least significant in the lowest. A digit above 9 raises.

	   # Examples

	   ```iecst
	   n := WORD_BCD_TO_UINT(WORD#16#0369);  // UINT#369
	   n := BYTE_BCD_TO_USINT(BYTE#16#25);   // USINT#25
	   ```
	*/
	FUNCTION BYTE_BCD_TO_USINT: USINT
		VAR_INPUT
			IN: BYTE;
		END_VAR
		VAR
			bcd: USINT;
			digit: USINT;
			place: USINT := 1;
		END_VAR
		{wasm 'nop' (params IN) (result bcd)}
		WHILE bcd > 0 DO
			digit := bcd MOD 16;
			IF digit > 9 THEN
				__RAISE('invalid BCD digit');
			END_IF;
			BYTE_BCD_TO_USINT := BYTE_BCD_TO_USINT + digit * place;
			place := place * 10;
			bcd := bcd / 16;
		END_WHILE;
	END_FUNCTION

	FUNCTION WORD_BCD_TO_UINT: UINT
		VAR_INPUT
			IN: WORD;
		END_VAR
		VAR
			bcd: UINT;
			digit: UINT;
			place: UINT := 1;
		END_VAR
		{wasm 'nop' (params IN) (result bcd)}
		WHILE bcd > 0 DO
			digit := bcd MOD 16;
			IF digit > 9 THEN
				__RAISE('invalid BCD digit');
			END_IF;
			WORD_BCD_TO_UINT := WORD_BCD_TO_UINT + digit * place;
			place := place * 10;
			bcd := bcd / 16;
		END_WHILE;
	END_FUNCTION

	FUNCTION DWORD_BCD_TO_UDINT: UDINT
		VAR_INPUT
			IN: DWORD;
		END_VAR
		VAR
			bcd: UDINT;
			digit: UDINT;
			place: UDINT := 1;
		END_VAR
		{wasm 'nop' (params IN) (result bcd)}
		WHILE bcd > 0 DO
			digit := bcd MOD 16;
			IF digit > 9 THEN
				__RAISE('invalid BCD digit');
			END_IF;
			DWORD_BCD_TO_UDINT := DWORD_BCD_TO_UDINT + digit * place;
			place := place * 10;
			bcd := bcd / 16;
		END_WHILE;
	END_FUNCTION

	FUNCTION LWORD_BCD_TO_ULINT: ULINT
		VAR_INPUT
			IN: LWORD;
		END_VAR
		VAR
			bcd: ULINT;
			digit: ULINT;
			place: ULINT := 1;
		END_VAR
		{wasm 'nop' (params IN) (result bcd)}
		WHILE bcd > 0 DO
			digit := bcd MOD 16;
			IF digit > 9 THEN
				__RAISE('invalid BCD digit');
			END_IF;
			LWORD_BCD_TO_ULINT := LWORD_BCD_TO_ULINT + digit * place;
			place := place * 10;
			bcd := bcd / 16;
		END_WHILE;
	END_FUNCTION

	/* Returns `IN` in BCD, one decimal digit in each 4 bits, the least
	   significant in the lowest. A number with more digits than the bit
	   string holds raises: more than 99 for a BYTE, 9999 for a WORD.

	   # Examples

	   ```iecst
	   w := UINT_TO_BCD_WORD(UINT#369);    // WORD#16#0369
	   b := USINT_TO_BCD_BYTE(USINT#25);   // BYTE#16#25
	   ```
	*/
	FUNCTION USINT_TO_BCD_BYTE: BYTE
		VAR_INPUT
			IN: USINT;
		END_VAR
		VAR
			value: USINT;
			bcd: USINT;
			place: USINT := 1;
		END_VAR
		IF IN > 99 THEN
			__RAISE('value too large for BCD');
		END_IF;
		value := IN;
		WHILE value > 0 DO
			bcd := bcd + (value MOD 10) * place;
			place := place * 16;
			value := value / 10;
		END_WHILE;
		{wasm 'nop' (params bcd) (result USINT_TO_BCD_BYTE)}
	END_FUNCTION

	FUNCTION UINT_TO_BCD_WORD: WORD
		VAR_INPUT
			IN: UINT;
		END_VAR
		VAR
			value: UINT;
			bcd: UINT;
			place: UINT := 1;
		END_VAR
		IF IN > 9999 THEN
			__RAISE('value too large for BCD');
		END_IF;
		value := IN;
		WHILE value > 0 DO
			bcd := bcd + (value MOD 10) * place;
			place := place * 16;
			value := value / 10;
		END_WHILE;
		{wasm 'nop' (params bcd) (result UINT_TO_BCD_WORD)}
	END_FUNCTION

	FUNCTION UDINT_TO_BCD_DWORD: DWORD
		VAR_INPUT
			IN: UDINT;
		END_VAR
		VAR
			value: UDINT;
			bcd: UDINT;
			place: UDINT := 1;
		END_VAR
		IF IN > 99999999 THEN
			__RAISE('value too large for BCD');
		END_IF;
		value := IN;
		WHILE value > 0 DO
			bcd := bcd + (value MOD 10) * place;
			place := place * 16;
			value := value / 10;
		END_WHILE;
		{wasm 'nop' (params bcd) (result UDINT_TO_BCD_DWORD)}
	END_FUNCTION

	FUNCTION ULINT_TO_BCD_LWORD: LWORD
		VAR_INPUT
			IN: ULINT;
		END_VAR
		VAR
			value: ULINT;
			bcd: ULINT;
			place: ULINT := 1;
		END_VAR
		IF IN > 9999999999999999 THEN
			__RAISE('value too large for BCD');
		END_IF;
		value := IN;
		WHILE value > 0 DO
			bcd := bcd + (value MOD 10) * place;
			place := place * 16;
			value := value / 10;
		END_WHILE;
		{wasm 'nop' (params bcd) (result ULINT_TO_BCD_LWORD)}
	END_FUNCTION

	/* The number `IN` holds in BCD, as `WORD_BCD_TO_UINT` and its siblings
	   give it, named by the result only.
	*/
	FUNCTION BCD_TO_USINT: USINT
		VAR_INPUT
			IN: BYTE;
		END_VAR
		BCD_TO_USINT := BYTE_BCD_TO_USINT(IN);
	END_FUNCTION

	FUNCTION BCD_TO_UINT: UINT
		VAR_INPUT
			IN: WORD;
		END_VAR
		BCD_TO_UINT := WORD_BCD_TO_UINT(IN);
	END_FUNCTION

	FUNCTION BCD_TO_UDINT: UDINT
		VAR_INPUT
			IN: DWORD;
		END_VAR
		BCD_TO_UDINT := DWORD_BCD_TO_UDINT(IN);
	END_FUNCTION

	FUNCTION BCD_TO_ULINT: ULINT
		VAR_INPUT
			IN: LWORD;
		END_VAR
		BCD_TO_ULINT := LWORD_BCD_TO_ULINT(IN);
	END_FUNCTION

	/* `IN` in BCD, as `UINT_TO_BCD_WORD` and its siblings give it, named by
	   the result only.
	*/
	FUNCTION TO_BCD_BYTE: BYTE
		VAR_INPUT
			IN: USINT;
		END_VAR
		TO_BCD_BYTE := USINT_TO_BCD_BYTE(IN);
	END_FUNCTION

	FUNCTION TO_BCD_WORD: WORD
		VAR_INPUT
			IN: UINT;
		END_VAR
		TO_BCD_WORD := UINT_TO_BCD_WORD(IN);
	END_FUNCTION

	FUNCTION TO_BCD_DWORD: DWORD
		VAR_INPUT
			IN: UDINT;
		END_VAR
		TO_BCD_DWORD := UDINT_TO_BCD_DWORD(IN);
	END_FUNCTION

	FUNCTION TO_BCD_LWORD: LWORD
		VAR_INPUT
			IN: ULINT;
		END_VAR
		TO_BCD_LWORD := ULINT_TO_BCD_LWORD(IN);
	END_FUNCTION

	/* Whether every 4 bits of `IN` hold a decimal digit, 0 to 9: whether
	   `IN` converts from BCD without raising.

	   # Examples

	   ```iecst
	   ok := IS_VALID_BCD(WORD#16#0369);  // TRUE
	   ok := IS_VALID_BCD(WORD#16#03A9);  // FALSE
	   ```
	*/
	FUNCTION IS_VALID_BCD: BOOL
		VAR_INPUT
			IN: BYTE;
		END_VAR
		VAR
			bcd: USINT;
		END_VAR
		{wasm 'nop' (params IN) (result bcd)}
		IS_VALID_BCD := TRUE;
		WHILE bcd > 0 DO
			IF bcd MOD 16 > 9 THEN
				IS_VALID_BCD := FALSE;
				RETURN;
			END_IF;
			bcd := bcd / 16;
		END_WHILE;
	END_FUNCTION

	FUNCTION IS_VALID_BCD: BOOL
		VAR_INPUT
			IN: WORD;
		END_VAR
		VAR
			bcd: UINT;
		END_VAR
		{wasm 'nop' (params IN) (result bcd)}
		IS_VALID_BCD := TRUE;
		WHILE bcd > 0 DO
			IF bcd MOD 16 > 9 THEN
				IS_VALID_BCD := FALSE;
				RETURN;
			END_IF;
			bcd := bcd / 16;
		END_WHILE;
	END_FUNCTION

	FUNCTION IS_VALID_BCD: BOOL
		VAR_INPUT
			IN: DWORD;
		END_VAR
		VAR
			bcd: UDINT;
		END_VAR
		{wasm 'nop' (params IN) (result bcd)}
		IS_VALID_BCD := TRUE;
		WHILE bcd > 0 DO
			IF bcd MOD 16 > 9 THEN
				IS_VALID_BCD := FALSE;
				RETURN;
			END_IF;
			bcd := bcd / 16;
		END_WHILE;
	END_FUNCTION

	FUNCTION IS_VALID_BCD: BOOL
		VAR_INPUT
			IN: LWORD;
		END_VAR
		VAR
			bcd: ULINT;
		END_VAR
		{wasm 'nop' (params IN) (result bcd)}
		IS_VALID_BCD := TRUE;
		WHILE bcd > 0 DO
			IF bcd MOD 16 > 9 THEN
				IS_VALID_BCD := FALSE;
				RETURN;
			END_IF;
			bcd := bcd / 16;
		END_WHILE;
	END_FUNCTION

	NAMESPACE Test
		USING Std.Unit
		USING Std.Convert

		{test}
		FUNCTION test_word ASSERT_EQ(TO_BIG_ENDIAN(WORD#16#1234), WORD#16#3412);
		END_FUNCTION

		{test}
		FUNCTION test_uint ASSERT_EQ(TO_BIG_ENDIAN(UINT#16#FF00), UINT#16#00FF);
		END_FUNCTION

		{test}
		FUNCTION test_int_keeps_its_sign ASSERT_EQ(TO_BIG_ENDIAN(INT#-2), INT#-257);
		END_FUNCTION

		{test}
		FUNCTION test_int_takes_a_sign ASSERT_EQ(TO_BIG_ENDIAN(INT#384), INT#-32767);
		END_FUNCTION

		{test}
		FUNCTION test_dword ASSERT_EQ(TO_BIG_ENDIAN(DWORD#16#12345678), DWORD#16#78563412);
		END_FUNCTION

		{test}
		FUNCTION test_dint ASSERT_EQ(TO_BIG_ENDIAN(DINT#-2), DINT#-16777217);
		END_FUNCTION

		{test}
		FUNCTION test_udint ASSERT_EQ(TO_BIG_ENDIAN(UDINT#16#11223344), UDINT#16#44332211);
		END_FUNCTION

		{test}
		FUNCTION test_lword ASSERT_EQ(TO_BIG_ENDIAN(LWORD#16#0102030405060708), LWORD#16#0807060504030201);
		END_FUNCTION

		{test}
		FUNCTION test_lint ASSERT_EQ(TO_BIG_ENDIAN(LINT#1), LINT#16#0100000000000000);
		END_FUNCTION

		{test}
		FUNCTION test_ulint ASSERT_EQ(TO_BIG_ENDIAN(ULINT#16#FF), ULINT#16#FF00000000000000);
		END_FUNCTION

		{test}
		FUNCTION test_real ASSERT_EQ(TO_BIG_ENDIAN(REAL#1.0), DWORD_TO_REAL(DWORD#16#0000803F));
		END_FUNCTION

		{test}
		FUNCTION test_lreal ASSERT_EQ(TO_BIG_ENDIAN(LREAL#1.0), LWORD_TO_LREAL(LWORD#16#000000000000F03F));
		END_FUNCTION

		{test}
		FUNCTION test_time ASSERT_EQ(TO_BIG_ENDIAN(T#1ms), T#16777216ms);
		END_FUNCTION

		{test}
		FUNCTION test_ltime ASSERT_EQ(TO_BIG_ENDIAN(LT#1ns), LT#72057594037927936ns);
		END_FUNCTION

		{test}
		FUNCTION test_one_byte ASSERT_EQ(TO_BIG_ENDIAN(BYTE#16#AB), BYTE#16#AB);
		END_FUNCTION

		{test}
		FUNCTION test_signed_byte ASSERT_EQ(FROM_BIG_ENDIAN(SINT#-3), SINT#-3);
		END_FUNCTION

		{test}
		FUNCTION test_round_trip_real ASSERT_EQ(FROM_BIG_ENDIAN(TO_BIG_ENDIAN(REAL#1.5)), REAL#1.5);
		END_FUNCTION

		{test}
		FUNCTION test_round_trip_dint ASSERT_EQ(FROM_BIG_ENDIAN(TO_BIG_ENDIAN(DINT#-123456)), DINT#-123456);
		END_FUNCTION

		{test}
		FUNCTION test_little_endian ASSERT_EQ(TO_LITTLE_ENDIAN(DWORD#16#12345678), DWORD#16#12345678);
		END_FUNCTION

		{test}
		FUNCTION test_from_little_endian ASSERT_EQ(FROM_LITTLE_ENDIAN(LINT#-5), LINT#-5);
		END_FUNCTION

		{test}
		FUNCTION test_bcd_byte ASSERT_EQ(USINT_TO_BCD_BYTE(USINT#25), BYTE#2#0010_0101);
		END_FUNCTION

		{test}
		FUNCTION test_bcd_word_decodes ASSERT_EQ(WORD_BCD_TO_UINT(WORD#2#0011_0110_1001), UINT#369);
		END_FUNCTION

		{test}
		FUNCTION test_bcd_dword ASSERT_EQ(UDINT_TO_BCD_DWORD(UDINT#12345678), DWORD#16#12345678);
		END_FUNCTION

		{test}
		FUNCTION test_bcd_lword_largest ASSERT_EQ(ULINT_TO_BCD_LWORD(ULINT#9999999999999999), LWORD#16#9999999999999999);
		END_FUNCTION

		{test}
		FUNCTION test_bcd_lword_decodes ASSERT_EQ(LWORD_BCD_TO_ULINT(LWORD#16#1234567890123456), ULINT#1234567890123456);
		END_FUNCTION

		{test}
		FUNCTION test_bcd_zero ASSERT_EQ(UINT_TO_BCD_WORD(UINT#0), WORD#0);
		END_FUNCTION

		{test}
		FUNCTION test_bcd_round_trip ASSERT_EQ(DWORD_BCD_TO_UDINT(UDINT_TO_BCD_DWORD(UDINT#99999999)), UDINT#99999999);
		END_FUNCTION

		{test}
		FUNCTION test_bcd_to_by_result ASSERT_EQ(BCD_TO_UINT(WORD#16#0042), UINT#42);
		END_FUNCTION

		{test}
		FUNCTION test_to_bcd_by_result ASSERT_EQ(TO_BCD_WORD(UINT#42), WORD#16#42);
		END_FUNCTION

		{test}
		FUNCTION test_valid_bcd ASSERT_EQ(IS_VALID_BCD(WORD#16#1234), TRUE);
		END_FUNCTION

		{test}
		FUNCTION test_invalid_bcd ASSERT_EQ(IS_VALID_BCD(WORD#16#12A4), FALSE);
		END_FUNCTION

		{test}
		FUNCTION test_invalid_bcd_top_digit ASSERT_EQ(IS_VALID_BCD(LWORD#16#F000000000000000), FALSE);
		END_FUNCTION

		{test}
		FUNCTION test_valid_bcd_byte ASSERT_EQ(IS_VALID_BCD(BYTE#16#99), TRUE);
		END_FUNCTION
	END_NAMESPACE
END_NAMESPACE

(* ---- Comparison.st ---- *)
/*
Comparison functions: the comparison operators under a name.

`GT`, `GE`, `EQ`, `LE` and `LT` compare each input with the next, however many
there are. `NE` compares two.

Each has one overload per elementary type. A `STRING` takes two, three or four
inputs, compared as the operators do.
*/
NAMESPACE Std.Comparison

	/* Returns `TRUE` when each input is greater than the next.

	   # Examples

	   ```iecst
	   b := GT(3, 2, 1);  // TRUE
	   b := GT(3, 3, 1);  // FALSE
	   ```
	*/
	FUNCTION GT: BOOL
		VAR_INPUT
			IN: BOOL...;
		END_VAR

		GT := ...IN>;
	END_FUNCTION

	FUNCTION GT: BOOL
		VAR_INPUT
			IN: SINT...;
		END_VAR

		GT := ...IN>;
	END_FUNCTION

	FUNCTION GT: BOOL
		VAR_INPUT
			IN: INT...;
		END_VAR

		GT := ...IN>;
	END_FUNCTION

	FUNCTION GT: BOOL
		VAR_INPUT
			IN: DINT...;
		END_VAR

		GT := ...IN>;
	END_FUNCTION

	FUNCTION GT: BOOL
		VAR_INPUT
			IN: LINT...;
		END_VAR

		GT := ...IN>;
	END_FUNCTION

	FUNCTION GT: BOOL
		VAR_INPUT
			IN: USINT...;
		END_VAR

		GT := ...IN>;
	END_FUNCTION

	FUNCTION GT: BOOL
		VAR_INPUT
			IN: UINT...;
		END_VAR

		GT := ...IN>;
	END_FUNCTION

	FUNCTION GT: BOOL
		VAR_INPUT
			IN: UDINT...;
		END_VAR

		GT := ...IN>;
	END_FUNCTION

	FUNCTION GT: BOOL
		VAR_INPUT
			IN: ULINT...;
		END_VAR

		GT := ...IN>;
	END_FUNCTION

	FUNCTION GT: BOOL
		VAR_INPUT
			IN: BYTE...;
		END_VAR

		GT := ...IN>;
	END_FUNCTION

	FUNCTION GT: BOOL
		VAR_INPUT
			IN: WORD...;
		END_VAR

		GT := ...IN>;
	END_FUNCTION

	FUNCTION GT: BOOL
		VAR_INPUT
			IN: DWORD...;
		END_VAR

		GT := ...IN>;
	END_FUNCTION

	FUNCTION GT: BOOL
		VAR_INPUT
			IN: LWORD...;
		END_VAR

		GT := ...IN>;
	END_FUNCTION

	FUNCTION GT: BOOL
		VAR_INPUT
			IN: REAL...;
		END_VAR

		GT := ...IN>;
	END_FUNCTION

	FUNCTION GT: BOOL
		VAR_INPUT
			IN: LREAL...;
		END_VAR

		GT := ...IN>;
	END_FUNCTION

	FUNCTION GT: BOOL
		VAR_INPUT
			IN1: STRING[255];
			IN2: STRING[255];
		END_VAR

		GT := IN1 > IN2;
	END_FUNCTION

	FUNCTION GT: BOOL
		VAR_INPUT
			IN1: STRING[255];
			IN2: STRING[255];
			IN3: STRING[255];
		END_VAR

		GT := IN1 > IN2 AND IN2 > IN3;
	END_FUNCTION

	FUNCTION GT: BOOL
		VAR_INPUT
			IN1: STRING[255];
			IN2: STRING[255];
			IN3: STRING[255];
			IN4: STRING[255];
		END_VAR

		GT := IN1 > IN2 AND IN2 > IN3 AND IN3 > IN4;
	END_FUNCTION

	FUNCTION GT: BOOL
		VAR_INPUT
			IN: TIME...;
		END_VAR

		GT := ...IN>;
	END_FUNCTION

	FUNCTION GT: BOOL
		VAR_INPUT
			IN: LTIME...;
		END_VAR

		GT := ...IN>;
	END_FUNCTION

	FUNCTION GT: BOOL
		VAR_INPUT
			IN: DATE...;
		END_VAR

		GT := ...IN>;
	END_FUNCTION

	FUNCTION GT: BOOL
		VAR_INPUT
			IN: LDATE...;
		END_VAR

		GT := ...IN>;
	END_FUNCTION

	FUNCTION GT: BOOL
		VAR_INPUT
			IN: TOD...;
		END_VAR

		GT := ...IN>;
	END_FUNCTION

	FUNCTION GT: BOOL
		VAR_INPUT
			IN: LTOD...;
		END_VAR

		GT := ...IN>;
	END_FUNCTION

	FUNCTION GT: BOOL
		VAR_INPUT
			IN: DT...;
		END_VAR

		GT := ...IN>;
	END_FUNCTION

	FUNCTION GT: BOOL
		VAR_INPUT
			IN: LDT...;
		END_VAR

		GT := ...IN>;
	END_FUNCTION

	FUNCTION GT: BOOL
		VAR_INPUT
			IN: CHAR...;
		END_VAR

		GT := ...IN>;
	END_FUNCTION

	/* Returns `TRUE` when each input is greater than or equal to the next.

	   # Examples

	   ```iecst
	   b := GE(3, 3, 1);  // TRUE
	   b := GE(1, 3, 3);  // FALSE
	   ```
	*/
	FUNCTION GE: BOOL
		VAR_INPUT
			IN: BOOL...;
		END_VAR

		GE := ...IN>=;
	END_FUNCTION

	FUNCTION GE: BOOL
		VAR_INPUT
			IN: SINT...;
		END_VAR

		GE := ...IN>=;
	END_FUNCTION

	FUNCTION GE: BOOL
		VAR_INPUT
			IN: INT...;
		END_VAR

		GE := ...IN>=;
	END_FUNCTION

	FUNCTION GE: BOOL
		VAR_INPUT
			IN: DINT...;
		END_VAR

		GE := ...IN>=;
	END_FUNCTION

	FUNCTION GE: BOOL
		VAR_INPUT
			IN: LINT...;
		END_VAR

		GE := ...IN>=;
	END_FUNCTION

	FUNCTION GE: BOOL
		VAR_INPUT
			IN: USINT...;
		END_VAR

		GE := ...IN>=;
	END_FUNCTION

	FUNCTION GE: BOOL
		VAR_INPUT
			IN: UINT...;
		END_VAR

		GE := ...IN>=;
	END_FUNCTION

	FUNCTION GE: BOOL
		VAR_INPUT
			IN: UDINT...;
		END_VAR

		GE := ...IN>=;
	END_FUNCTION

	FUNCTION GE: BOOL
		VAR_INPUT
			IN: ULINT...;
		END_VAR

		GE := ...IN>=;
	END_FUNCTION

	FUNCTION GE: BOOL
		VAR_INPUT
			IN: BYTE...;
		END_VAR

		GE := ...IN>=;
	END_FUNCTION

	FUNCTION GE: BOOL
		VAR_INPUT
			IN: WORD...;
		END_VAR

		GE := ...IN>=;
	END_FUNCTION

	FUNCTION GE: BOOL
		VAR_INPUT
			IN: DWORD...;
		END_VAR

		GE := ...IN>=;
	END_FUNCTION

	FUNCTION GE: BOOL
		VAR_INPUT
			IN: LWORD...;
		END_VAR

		GE := ...IN>=;
	END_FUNCTION

	FUNCTION GE: BOOL
		VAR_INPUT
			IN: REAL...;
		END_VAR

		GE := ...IN>=;
	END_FUNCTION

	FUNCTION GE: BOOL
		VAR_INPUT
			IN: LREAL...;
		END_VAR

		GE := ...IN>=;
	END_FUNCTION

	FUNCTION GE: BOOL
		VAR_INPUT
			IN1: STRING[255];
			IN2: STRING[255];
		END_VAR

		GE := IN1 >= IN2;
	END_FUNCTION

	FUNCTION GE: BOOL
		VAR_INPUT
			IN1: STRING[255];
			IN2: STRING[255];
			IN3: STRING[255];
		END_VAR

		GE := IN1 >= IN2 AND IN2 >= IN3;
	END_FUNCTION

	FUNCTION GE: BOOL
		VAR_INPUT
			IN1: STRING[255];
			IN2: STRING[255];
			IN3: STRING[255];
			IN4: STRING[255];
		END_VAR

		GE := IN1 >= IN2 AND IN2 >= IN3 AND IN3 >= IN4;
	END_FUNCTION

	FUNCTION GE: BOOL
		VAR_INPUT
			IN: TIME...;
		END_VAR

		GE := ...IN>=;
	END_FUNCTION

	FUNCTION GE: BOOL
		VAR_INPUT
			IN: LTIME...;
		END_VAR

		GE := ...IN>=;
	END_FUNCTION

	FUNCTION GE: BOOL
		VAR_INPUT
			IN: DATE...;
		END_VAR

		GE := ...IN>=;
	END_FUNCTION

	FUNCTION GE: BOOL
		VAR_INPUT
			IN: LDATE...;
		END_VAR

		GE := ...IN>=;
	END_FUNCTION

	FUNCTION GE: BOOL
		VAR_INPUT
			IN: TOD...;
		END_VAR

		GE := ...IN>=;
	END_FUNCTION

	FUNCTION GE: BOOL
		VAR_INPUT
			IN: LTOD...;
		END_VAR

		GE := ...IN>=;
	END_FUNCTION

	FUNCTION GE: BOOL
		VAR_INPUT
			IN: DT...;
		END_VAR

		GE := ...IN>=;
	END_FUNCTION

	FUNCTION GE: BOOL
		VAR_INPUT
			IN: LDT...;
		END_VAR

		GE := ...IN>=;
	END_FUNCTION

	FUNCTION GE: BOOL
		VAR_INPUT
			IN: CHAR...;
		END_VAR

		GE := ...IN>=;
	END_FUNCTION

	/* Returns `TRUE` when its inputs are all equal.

	   # Examples

	   ```iecst
	   b := EQ(2, 2, 2);  // TRUE
	   b := EQ(2, 2, 3);  // FALSE
	   ```
	*/
	FUNCTION EQ: BOOL
		VAR_INPUT
			IN: BOOL...;
		END_VAR

		EQ := ...IN=;
	END_FUNCTION

	FUNCTION EQ: BOOL
		VAR_INPUT
			IN: SINT...;
		END_VAR

		EQ := ...IN=;
	END_FUNCTION

	FUNCTION EQ: BOOL
		VAR_INPUT
			IN: INT...;
		END_VAR

		EQ := ...IN=;
	END_FUNCTION

	FUNCTION EQ: BOOL
		VAR_INPUT
			IN: DINT...;
		END_VAR

		EQ := ...IN=;
	END_FUNCTION

	FUNCTION EQ: BOOL
		VAR_INPUT
			IN: LINT...;
		END_VAR

		EQ := ...IN=;
	END_FUNCTION

	FUNCTION EQ: BOOL
		VAR_INPUT
			IN: USINT...;
		END_VAR

		EQ := ...IN=;
	END_FUNCTION

	FUNCTION EQ: BOOL
		VAR_INPUT
			IN: UINT...;
		END_VAR

		EQ := ...IN=;
	END_FUNCTION

	FUNCTION EQ: BOOL
		VAR_INPUT
			IN: UDINT...;
		END_VAR

		EQ := ...IN=;
	END_FUNCTION

	FUNCTION EQ: BOOL
		VAR_INPUT
			IN: ULINT...;
		END_VAR

		EQ := ...IN=;
	END_FUNCTION

	FUNCTION EQ: BOOL
		VAR_INPUT
			IN: BYTE...;
		END_VAR

		EQ := ...IN=;
	END_FUNCTION

	FUNCTION EQ: BOOL
		VAR_INPUT
			IN: WORD...;
		END_VAR

		EQ := ...IN=;
	END_FUNCTION

	FUNCTION EQ: BOOL
		VAR_INPUT
			IN: DWORD...;
		END_VAR

		EQ := ...IN=;
	END_FUNCTION

	FUNCTION EQ: BOOL
		VAR_INPUT
			IN: LWORD...;
		END_VAR

		EQ := ...IN=;
	END_FUNCTION

	FUNCTION EQ: BOOL
		VAR_INPUT
			IN: REAL...;
		END_VAR

		EQ := ...IN=;
	END_FUNCTION

	FUNCTION EQ: BOOL
		VAR_INPUT
			IN: LREAL...;
		END_VAR

		EQ := ...IN=;
	END_FUNCTION

	FUNCTION EQ: BOOL
		VAR_INPUT
			IN1: STRING[255];
			IN2: STRING[255];
		END_VAR

		EQ := IN1 = IN2;
	END_FUNCTION

	FUNCTION EQ: BOOL
		VAR_INPUT
			IN1: STRING[255];
			IN2: STRING[255];
			IN3: STRING[255];
		END_VAR

		EQ := IN1 = IN2 AND IN2 = IN3;
	END_FUNCTION

	FUNCTION EQ: BOOL
		VAR_INPUT
			IN1: STRING[255];
			IN2: STRING[255];
			IN3: STRING[255];
			IN4: STRING[255];
		END_VAR

		EQ := IN1 = IN2 AND IN2 = IN3 AND IN3 = IN4;
	END_FUNCTION

	FUNCTION EQ: BOOL
		VAR_INPUT
			IN: TIME...;
		END_VAR

		EQ := ...IN=;
	END_FUNCTION

	FUNCTION EQ: BOOL
		VAR_INPUT
			IN: LTIME...;
		END_VAR

		EQ := ...IN=;
	END_FUNCTION

	FUNCTION EQ: BOOL
		VAR_INPUT
			IN: DATE...;
		END_VAR

		EQ := ...IN=;
	END_FUNCTION

	FUNCTION EQ: BOOL
		VAR_INPUT
			IN: LDATE...;
		END_VAR

		EQ := ...IN=;
	END_FUNCTION

	FUNCTION EQ: BOOL
		VAR_INPUT
			IN: TOD...;
		END_VAR

		EQ := ...IN=;
	END_FUNCTION

	FUNCTION EQ: BOOL
		VAR_INPUT
			IN: LTOD...;
		END_VAR

		EQ := ...IN=;
	END_FUNCTION

	FUNCTION EQ: BOOL
		VAR_INPUT
			IN: DT...;
		END_VAR

		EQ := ...IN=;
	END_FUNCTION

	FUNCTION EQ: BOOL
		VAR_INPUT
			IN: LDT...;
		END_VAR

		EQ := ...IN=;
	END_FUNCTION

	FUNCTION EQ: BOOL
		VAR_INPUT
			IN: CHAR...;
		END_VAR

		EQ := ...IN=;
	END_FUNCTION

	/* Returns `TRUE` when each input is less than or equal to the next.

	   # Examples

	   ```iecst
	   b := LE(1, 3, 3);  // TRUE
	   b := LE(3, 3, 1);  // FALSE
	   ```
	*/
	FUNCTION LE: BOOL
		VAR_INPUT
			IN: BOOL...;
		END_VAR

		LE := ...IN<=;
	END_FUNCTION

	FUNCTION LE: BOOL
		VAR_INPUT
			IN: SINT...;
		END_VAR

		LE := ...IN<=;
	END_FUNCTION

	FUNCTION LE: BOOL
		VAR_INPUT
			IN: INT...;
		END_VAR

		LE := ...IN<=;
	END_FUNCTION

	FUNCTION LE: BOOL
		VAR_INPUT
			IN: DINT...;
		END_VAR

		LE := ...IN<=;
	END_FUNCTION

	FUNCTION LE: BOOL
		VAR_INPUT
			IN: LINT...;
		END_VAR

		LE := ...IN<=;
	END_FUNCTION

	FUNCTION LE: BOOL
		VAR_INPUT
			IN: USINT...;
		END_VAR

		LE := ...IN<=;
	END_FUNCTION

	FUNCTION LE: BOOL
		VAR_INPUT
			IN: UINT...;
		END_VAR

		LE := ...IN<=;
	END_FUNCTION

	FUNCTION LE: BOOL
		VAR_INPUT
			IN: UDINT...;
		END_VAR

		LE := ...IN<=;
	END_FUNCTION

	FUNCTION LE: BOOL
		VAR_INPUT
			IN: ULINT...;
		END_VAR

		LE := ...IN<=;
	END_FUNCTION

	FUNCTION LE: BOOL
		VAR_INPUT
			IN: BYTE...;
		END_VAR

		LE := ...IN<=;
	END_FUNCTION

	FUNCTION LE: BOOL
		VAR_INPUT
			IN: WORD...;
		END_VAR

		LE := ...IN<=;
	END_FUNCTION

	FUNCTION LE: BOOL
		VAR_INPUT
			IN: DWORD...;
		END_VAR

		LE := ...IN<=;
	END_FUNCTION

	FUNCTION LE: BOOL
		VAR_INPUT
			IN: LWORD...;
		END_VAR

		LE := ...IN<=;
	END_FUNCTION

	FUNCTION LE: BOOL
		VAR_INPUT
			IN: REAL...;
		END_VAR

		LE := ...IN<=;
	END_FUNCTION

	FUNCTION LE: BOOL
		VAR_INPUT
			IN: LREAL...;
		END_VAR

		LE := ...IN<=;
	END_FUNCTION

	FUNCTION LE: BOOL
		VAR_INPUT
			IN1: STRING[255];
			IN2: STRING[255];
		END_VAR

		LE := IN1 <= IN2;
	END_FUNCTION

	FUNCTION LE: BOOL
		VAR_INPUT
			IN1: STRING[255];
			IN2: STRING[255];
			IN3: STRING[255];
		END_VAR

		LE := IN1 <= IN2 AND IN2 <= IN3;
	END_FUNCTION

	FUNCTION LE: BOOL
		VAR_INPUT
			IN1: STRING[255];
			IN2: STRING[255];
			IN3: STRING[255];
			IN4: STRING[255];
		END_VAR

		LE := IN1 <= IN2 AND IN2 <= IN3 AND IN3 <= IN4;
	END_FUNCTION

	FUNCTION LE: BOOL
		VAR_INPUT
			IN: TIME...;
		END_VAR

		LE := ...IN<=;
	END_FUNCTION

	FUNCTION LE: BOOL
		VAR_INPUT
			IN: LTIME...;
		END_VAR

		LE := ...IN<=;
	END_FUNCTION

	FUNCTION LE: BOOL
		VAR_INPUT
			IN: DATE...;
		END_VAR

		LE := ...IN<=;
	END_FUNCTION

	FUNCTION LE: BOOL
		VAR_INPUT
			IN: LDATE...;
		END_VAR

		LE := ...IN<=;
	END_FUNCTION

	FUNCTION LE: BOOL
		VAR_INPUT
			IN: TOD...;
		END_VAR

		LE := ...IN<=;
	END_FUNCTION

	FUNCTION LE: BOOL
		VAR_INPUT
			IN: LTOD...;
		END_VAR

		LE := ...IN<=;
	END_FUNCTION

	FUNCTION LE: BOOL
		VAR_INPUT
			IN: DT...;
		END_VAR

		LE := ...IN<=;
	END_FUNCTION

	FUNCTION LE: BOOL
		VAR_INPUT
			IN: LDT...;
		END_VAR

		LE := ...IN<=;
	END_FUNCTION

	FUNCTION LE: BOOL
		VAR_INPUT
			IN: CHAR...;
		END_VAR

		LE := ...IN<=;
	END_FUNCTION

	/* Returns `TRUE` when each input is less than the next.

	   # Examples

	   ```iecst
	   b := LT(1, 2, 3);  // TRUE
	   b := LT(1, 3, 3);  // FALSE
	   ```
	*/
	FUNCTION LT: BOOL
		VAR_INPUT
			IN: BOOL...;
		END_VAR

		LT := ...IN<;
	END_FUNCTION

	FUNCTION LT: BOOL
		VAR_INPUT
			IN: SINT...;
		END_VAR

		LT := ...IN<;
	END_FUNCTION

	FUNCTION LT: BOOL
		VAR_INPUT
			IN: INT...;
		END_VAR

		LT := ...IN<;
	END_FUNCTION

	FUNCTION LT: BOOL
		VAR_INPUT
			IN: DINT...;
		END_VAR

		LT := ...IN<;
	END_FUNCTION

	FUNCTION LT: BOOL
		VAR_INPUT
			IN: LINT...;
		END_VAR

		LT := ...IN<;
	END_FUNCTION

	FUNCTION LT: BOOL
		VAR_INPUT
			IN: USINT...;
		END_VAR

		LT := ...IN<;
	END_FUNCTION

	FUNCTION LT: BOOL
		VAR_INPUT
			IN: UINT...;
		END_VAR

		LT := ...IN<;
	END_FUNCTION

	FUNCTION LT: BOOL
		VAR_INPUT
			IN: UDINT...;
		END_VAR

		LT := ...IN<;
	END_FUNCTION

	FUNCTION LT: BOOL
		VAR_INPUT
			IN: ULINT...;
		END_VAR

		LT := ...IN<;
	END_FUNCTION

	FUNCTION LT: BOOL
		VAR_INPUT
			IN: BYTE...;
		END_VAR

		LT := ...IN<;
	END_FUNCTION

	FUNCTION LT: BOOL
		VAR_INPUT
			IN: WORD...;
		END_VAR

		LT := ...IN<;
	END_FUNCTION

	FUNCTION LT: BOOL
		VAR_INPUT
			IN: DWORD...;
		END_VAR

		LT := ...IN<;
	END_FUNCTION

	FUNCTION LT: BOOL
		VAR_INPUT
			IN: LWORD...;
		END_VAR

		LT := ...IN<;
	END_FUNCTION

	FUNCTION LT: BOOL
		VAR_INPUT
			IN: REAL...;
		END_VAR

		LT := ...IN<;
	END_FUNCTION

	FUNCTION LT: BOOL
		VAR_INPUT
			IN: LREAL...;
		END_VAR

		LT := ...IN<;
	END_FUNCTION

	FUNCTION LT: BOOL
		VAR_INPUT
			IN1: STRING[255];
			IN2: STRING[255];
		END_VAR

		LT := IN1 < IN2;
	END_FUNCTION

	FUNCTION LT: BOOL
		VAR_INPUT
			IN1: STRING[255];
			IN2: STRING[255];
			IN3: STRING[255];
		END_VAR

		LT := IN1 < IN2 AND IN2 < IN3;
	END_FUNCTION

	FUNCTION LT: BOOL
		VAR_INPUT
			IN1: STRING[255];
			IN2: STRING[255];
			IN3: STRING[255];
			IN4: STRING[255];
		END_VAR

		LT := IN1 < IN2 AND IN2 < IN3 AND IN3 < IN4;
	END_FUNCTION

	FUNCTION LT: BOOL
		VAR_INPUT
			IN: TIME...;
		END_VAR

		LT := ...IN<;
	END_FUNCTION

	FUNCTION LT: BOOL
		VAR_INPUT
			IN: LTIME...;
		END_VAR

		LT := ...IN<;
	END_FUNCTION

	FUNCTION LT: BOOL
		VAR_INPUT
			IN: DATE...;
		END_VAR

		LT := ...IN<;
	END_FUNCTION

	FUNCTION LT: BOOL
		VAR_INPUT
			IN: LDATE...;
		END_VAR

		LT := ...IN<;
	END_FUNCTION

	FUNCTION LT: BOOL
		VAR_INPUT
			IN: TOD...;
		END_VAR

		LT := ...IN<;
	END_FUNCTION

	FUNCTION LT: BOOL
		VAR_INPUT
			IN: LTOD...;
		END_VAR

		LT := ...IN<;
	END_FUNCTION

	FUNCTION LT: BOOL
		VAR_INPUT
			IN: DT...;
		END_VAR

		LT := ...IN<;
	END_FUNCTION

	FUNCTION LT: BOOL
		VAR_INPUT
			IN: LDT...;
		END_VAR

		LT := ...IN<;
	END_FUNCTION

	FUNCTION LT: BOOL
		VAR_INPUT
			IN: CHAR...;
		END_VAR

		LT := ...IN<;
	END_FUNCTION

	/* Returns `TRUE` when `IN1` and `IN2` differ.

	   # Examples

	   ```iecst
	   b := NE(1, 2);  // TRUE
	   b := NE(2, 2);  // FALSE
	   ```
	*/
	FUNCTION NE: BOOL
		VAR_INPUT
			IN1: BOOL;
			IN2: BOOL;
		END_VAR

		NE := IN1 <> IN2;
	END_FUNCTION

	FUNCTION NE: BOOL
		VAR_INPUT
			IN1: SINT;
			IN2: SINT;
		END_VAR

		NE := IN1 <> IN2;
	END_FUNCTION

	FUNCTION NE: BOOL
		VAR_INPUT
			IN1: INT;
			IN2: INT;
		END_VAR

		NE := IN1 <> IN2;
	END_FUNCTION

	FUNCTION NE: BOOL
		VAR_INPUT
			IN1: DINT;
			IN2: DINT;
		END_VAR

		NE := IN1 <> IN2;
	END_FUNCTION

	FUNCTION NE: BOOL
		VAR_INPUT
			IN1: LINT;
			IN2: LINT;
		END_VAR

		NE := IN1 <> IN2;
	END_FUNCTION

	FUNCTION NE: BOOL
		VAR_INPUT
			IN1: USINT;
			IN2: USINT;
		END_VAR

		NE := IN1 <> IN2;
	END_FUNCTION

	FUNCTION NE: BOOL
		VAR_INPUT
			IN1: UINT;
			IN2: UINT;
		END_VAR

		NE := IN1 <> IN2;
	END_FUNCTION

	FUNCTION NE: BOOL
		VAR_INPUT
			IN1: UDINT;
			IN2: UDINT;
		END_VAR

		NE := IN1 <> IN2;
	END_FUNCTION

	FUNCTION NE: BOOL
		VAR_INPUT
			IN1: ULINT;
			IN2: ULINT;
		END_VAR

		NE := IN1 <> IN2;
	END_FUNCTION

	FUNCTION NE: BOOL
		VAR_INPUT
			IN1: BYTE;
			IN2: BYTE;
		END_VAR

		NE := IN1 <> IN2;
	END_FUNCTION

	FUNCTION NE: BOOL
		VAR_INPUT
			IN1: WORD;
			IN2: WORD;
		END_VAR

		NE := IN1 <> IN2;
	END_FUNCTION

	FUNCTION NE: BOOL
		VAR_INPUT
			IN1: DWORD;
			IN2: DWORD;
		END_VAR

		NE := IN1 <> IN2;
	END_FUNCTION

	FUNCTION NE: BOOL
		VAR_INPUT
			IN1: LWORD;
			IN2: LWORD;
		END_VAR

		NE := IN1 <> IN2;
	END_FUNCTION

	{allow 'float-equality'}
	FUNCTION NE: BOOL
		VAR_INPUT
			IN1: REAL;
			IN2: REAL;
		END_VAR

		NE := IN1 <> IN2;
	END_FUNCTION

	{allow 'float-equality'}
	FUNCTION NE: BOOL
		VAR_INPUT
			IN1: LREAL;
			IN2: LREAL;
		END_VAR

		NE := IN1 <> IN2;
	END_FUNCTION

	FUNCTION NE: BOOL
		VAR_INPUT
			IN1: TIME;
			IN2: TIME;
		END_VAR

		NE := IN1 <> IN2;
	END_FUNCTION

	FUNCTION NE: BOOL
		VAR_INPUT
			IN1: LTIME;
			IN2: LTIME;
		END_VAR

		NE := IN1 <> IN2;
	END_FUNCTION

	FUNCTION NE: BOOL
		VAR_INPUT
			IN1: DATE;
			IN2: DATE;
		END_VAR

		NE := IN1 <> IN2;
	END_FUNCTION

	FUNCTION NE: BOOL
		VAR_INPUT
			IN1: LDATE;
			IN2: LDATE;
		END_VAR

		NE := IN1 <> IN2;
	END_FUNCTION

	FUNCTION NE: BOOL
		VAR_INPUT
			IN1: TOD;
			IN2: TOD;
		END_VAR

		NE := IN1 <> IN2;
	END_FUNCTION

	FUNCTION NE: BOOL
		VAR_INPUT
			IN1: LTOD;
			IN2: LTOD;
		END_VAR

		NE := IN1 <> IN2;
	END_FUNCTION

	FUNCTION NE: BOOL
		VAR_INPUT
			IN1: DT;
			IN2: DT;
		END_VAR

		NE := IN1 <> IN2;
	END_FUNCTION

	FUNCTION NE: BOOL
		VAR_INPUT
			IN1: LDT;
			IN2: LDT;
		END_VAR

		NE := IN1 <> IN2;
	END_FUNCTION

	FUNCTION NE: BOOL
		VAR_INPUT
			IN1: CHAR;
			IN2: CHAR;
		END_VAR

		NE := IN1 <> IN2;
	END_FUNCTION

	FUNCTION NE: BOOL
		VAR_INPUT
			IN1: STRING[255];
			IN2: STRING[255];
		END_VAR

		NE := IN1 <> IN2;
	END_FUNCTION

	NAMESPACE Test
		USING Std.Unit

		{test}
		FUNCTION test_gt
			ASSERT(GT(3, 2, 1));
			ASSERT(NOT GT(3, 3, 1));
		END_FUNCTION

		{test}
		FUNCTION test_ge
			ASSERT(GE(3, 3, 1));
			ASSERT(NOT GE(1, 3, 3));
		END_FUNCTION

		{test}
		FUNCTION test_eq
			ASSERT(EQ(2, 2, 2));
			ASSERT(NOT EQ(2, 2, 3));
		END_FUNCTION

		{test}
		FUNCTION test_le
			ASSERT(LE(1, 3, 3));
			ASSERT(NOT LE(3, 3, 1));
		END_FUNCTION

		{test}
		FUNCTION test_lt
			ASSERT(LT(1, 2, 3));
			ASSERT(NOT LT(1, 3, 3));
		END_FUNCTION

		{test}
		FUNCTION test_ne
			ASSERT(NE(1, 2));
			ASSERT(NOT NE(2, 2));
		END_FUNCTION
	END_NAMESPACE
END_NAMESPACE
